ABB RobotStudio station: welding_of_volumetric_parts.rsstn

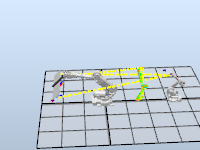
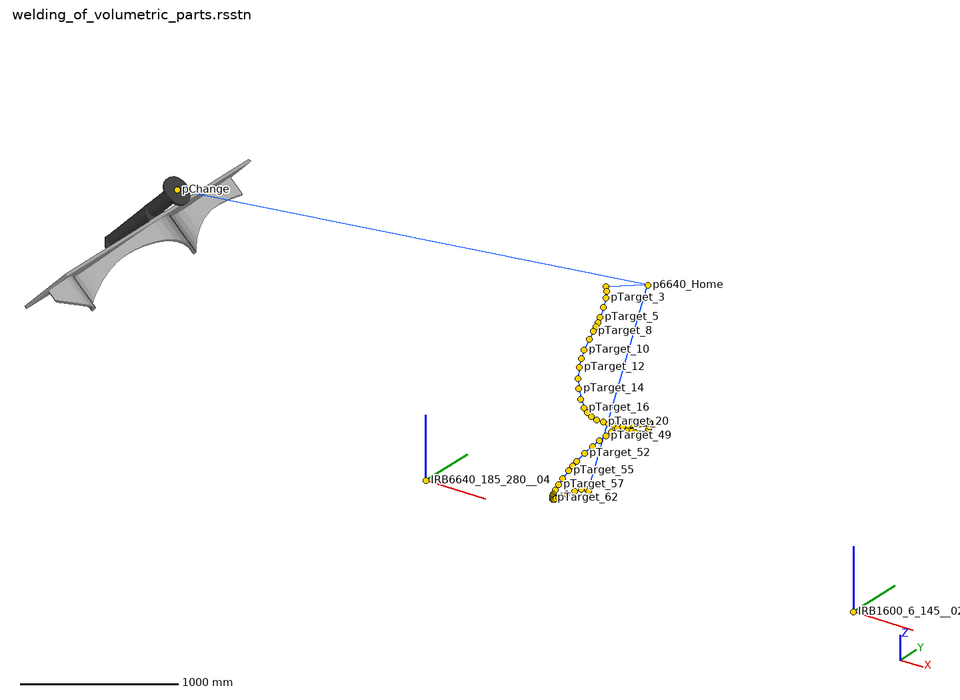
[picture v1: parts stored in the station drawn from their meshes, with robot base, taught points and paths (robot models come from the ABB library and are not in the file)]
Station Station (saved by RobotStudio 21.2.9526.0)
Controller Controller_LR, task T_ROB2: task frame (RAPID world) sits at (3300, 0, 0) mm, rotated rx 0 ry 0 rz 180 deg in the station
Controller Controller_LR, task T_ROB1: task frame (RAPID world) sits at (3300, 0, 0) mm, rotated rx 0 ry 0 rz 180 deg in the station
Controller Controller_LR
  mechanical unit ROB_1: IRB6640_185_280__04, 6 joints, base frame (3300, 0, 0) mm, rotated rx 0 ry 0 rz 180 deg
  mechanical unit ROB_2: IRB1600_6_145__02, 6 joints, base frame (0, 0, 0) mm
Layout (positions relative to the parent item):
  - IRB1600_6_145__02 [mechanism, from Robots\IRB1600_6_145_G_02.rslib] at (3300, 0, 0) mm, rotated rx 0 ry 0 rz 180 deg; joint values [0, -0.6981, 0, 0, 0.4363, 3.1416] (rad or m)
  - IRB6640_185_280__04 [mechanism, from Robots\IRB6640_185_280_G_04.rslib] at (0, 0, 0) mm; joint values [0, -0.6981, -2.2689, 0, -0.9599, 0] (rad or m)
  - training_part1 [part] at (-1918.49, 0, 1506.92) mm, rotated rx 180 ry -45 rz -180 deg, size 449.3 x 2022.8 x 720 mm
  - Binzel_air_22 [mechanism, from Tools\Binzel_air_22.rslib] at (3077.54, 0, 1425.23) mm, rotated rx 0 ry -75 rz 0 deg
Attachment: training_part1 is attached to IRB6640_185_280__04 / Link6
Attachment: Binzel_air_22 is attached to IRB1600_6_145__02 / Link6
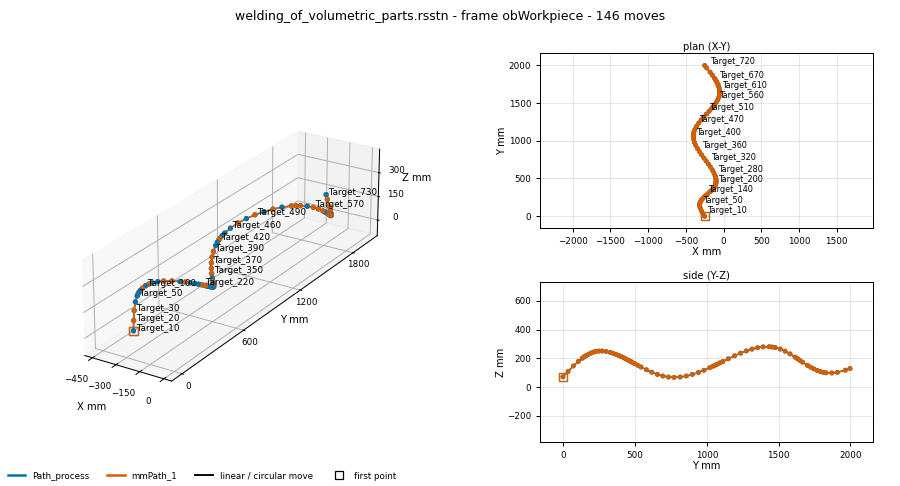
[picture p0: tool path of welding_of_volumetric_parts.rsstn in frame obWorkpiece, 146 of 224 moves have a stored position in this frame; points joined in program order, loops and branches not executed]
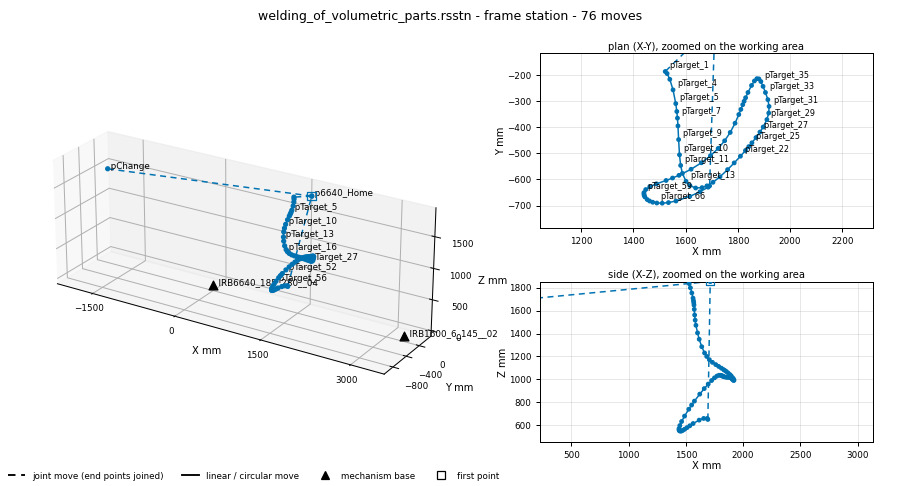
[picture p1: tool path of welding_of_volumetric_parts.rsstn in frame station, 76 of 224 moves have a stored position in this frame; points joined in program order, loops and branches not executed]
Targets, tools, work objects and paths stored in the station, written as RAPID:
! task T_ROB1
MODULE Module1
  VAR SyncIdent Ident_1;
  VAR SyncIdent Ident_2;
  PERS Tasks Task_1{2}:=[["T_ROB1"],["T_ROB2"]];
  CONST robtarget pTarget_1:=[[1778.181697527,186.200299858,1862.655645301],[0.542148406,0.793411995,0.256756469,-0.103192188],[-1,0,-1,0],[9E+09,9E+09,9E+09,9E+09,9E+09,9E+09]];
  CONST robtarget pTarget_2:=[[1770.994188299,194.050467885,1836.295876308],[0.547547156,0.793734178,0.24715111,-0.095365067],[-1,0,-1,0],[9E+09,9E+09,9E+09,9E+09,9E+09,9E+09]];
  CONST robtarget pTarget_3:=[[1760.652825255,216.161560279,1800.133289507],[0.558555641,0.792378,0.228049318,-0.090256356],[-1,0,-1,0],[9E+09,9E+09,9E+09,9E+09,9E+09,9E+09]];
  CONST robtarget pTarget_4:=[[1748.290299895,256.657627996,1755.126396139],[0.576885547,0.787168315,0.198285168,-0.090841082],[-1,0,-1,0],[9E+09,9E+09,9E+09,9E+09,9E+09,9E+09]];
  CONST robtarget pTarget_5:=[[1737.829387141,309.266346265,1710.003660644],[0.600170273,0.776755771,0.163693874,-0.098236606],[-1,0,-1,0],[9E+09,9E+09,9E+09,9E+09,9E+09,9E+09]];
  CONST robtarget pTarget_6:=[[1733.804937068,339.397116728,1687.439781271],[0.613523349,0.769208972,0.145104916,-0.104169199],[-1,0,-1,0],[9E+09,9E+09,9E+09,9E+09,9E+09,9E+09]];
  CONST robtarget pTarget_7:=[[1731.345474568,364.887069734,1669.469926767],[0.624865432,0.761982746,0.12988239,-0.109800051],[-1,0,-1,0],[9E+09,9E+09,9E+09,9E+09,9E+09,9E+09]];
  CONST robtarget pTarget_8:=[[1729.439217622,394.798254229,1649.227463455],[0.638246376,0.752542699,0.112494045,-0.116902268],[-1,0,-1,0],[9E+09,9E+09,9E+09,9E+09,9E+09,9E+09]];
  CONST robtarget pTarget_9:=[[1726.894203356,447.184397046,1611.766562004],[0.661982515,0.733744338,0.082051113,-0.129096907],[-1,0,-1,0],[9E+09,9E+09,9E+09,9E+09,9E+09,9E+09]];
  CONST robtarget pTarget_10:=[[1723.544484943,505.45769037,1562.230464943],[0.689273971,0.709178686,0.04680241,-0.140629006],[-1,0,-1,0],[9E+09,9E+09,9E+09,9E+09,9E+09,9E+09]];
  CONST robtarget pTarget_11:=[[1719.097770684,546.281247526,1517.405345945],[0.709465359,0.689213309,0.019587314,-0.145808972],[-1,0,-1,0],[9E+09,9E+09,9E+09,9E+09,9E+09,9E+09]];
  CONST robtarget pTarget_12:=[[1712.357728352,576.685538105,1472.436688768],[0.725592454,0.672374376,-0.004172996,-0.146324552],[-1,0,-1,0],[9E+09,9E+09,9E+09,9E+09,9E+09,9E+09]];
  CONST robtarget pTarget_13:=[[1698.481718308,607.168067285,1406.157920867],[0.743150521,0.65316553,-0.03513516,-0.140952521],[-1,1,-1,0],[9E+09,9E+09,9E+09,9E+09,9E+09,9E+09]];
  CONST robtarget pTarget_14:=[[1683.689245608,623.318514853,1350.511714032],[0.752710379,0.642114247,-0.059185356,-0.132715759],[-1,1,-1,0],[9E+09,9E+09,9E+09,9E+09,9E+09,9E+09]];
  CONST robtarget pTarget_15:=[[1661.611102892,632.661072606,1285.206196443],[0.756964574,0.636483122,-0.086573404,-0.119995478],[-1,1,-1,0],[9E+09,9E+09,9E+09,9E+09,9E+09,9E+09]];
  CONST robtarget pTarget_16:=[[1636.974570689,631.269638782,1230.880629936],[0.752461483,0.640504386,-0.109446392,-0.107598031],[-1,1,-1,0],[9E+09,9E+09,9E+09,9E+09,9E+09,9E+09]];
  CONST robtarget pTarget_17:=[[1618.266585822,624.412772296,1200.303251277],[0.744570861,0.648569679,-0.122376791,-0.099977627],[-1,1,-1,0],[9E+09,9E+09,9E+09,9E+09,9E+09,9E+09]];
  CONST robtarget pTarget_18:=[[1595.31025739,610.899403989,1172.356577935],[0.73138813,0.662260205,-0.133827929,-0.092590006],[-1,0,-1,0],[9E+09,9E+09,9E+09,9E+09,9E+09,9E+09]];
  CONST robtarget pTarget_19:=[[1568.252391964,589.541208244,1148.621347281],[0.712476477,0.681687181,-0.142360657,-0.086100519],[-1,0,-1,0],[9E+09,9E+09,9E+09,9E+09,9E+09,9E+09]];
  CONST robtarget pTarget_20:=[[1539.248164994,562.206507767,1129.084627739],[0.689417374,0.704583469,-0.14724324,-0.081149543],[-1,0,-1,0],[9E+09,9E+09,9E+09,9E+09,9E+09,9E+09]];
  CONST robtarget pTarget_21:=[[1513.907722067,536.515023967,1113.043516835],[0.667709522,0.725077896,-0.149409413,-0.078120848],[-1,0,-1,0],[9E+09,9E+09,9E+09,9E+09,9E+09,9E+09]];
  CONST robtarget pTarget_22:=[[1490.06843077,510.919096367,1097.932249558],[0.645797019,0.744781689,-0.14976235,-0.076273744],[-1,0,-1,0],[9E+09,9E+09,9E+09,9E+09,9E+09,9E+09]];
  CONST robtarget pTarget_23:=[[1470.694976412,489.03192048,1085.160534616],[0.626718168,0.761182635,-0.148768738,-0.075453277],[-1,0,-1,0],[9E+09,9E+09,9E+09,9E+09,9E+09,9E+09]];
  CONST robtarget pTarget_24:=[[1458.007723014,474.098201767,1076.33725701],[0.613483711,0.772169291,-0.1474183,-0.075234082],[-1,0,-1,0],[9E+09,9E+09,9E+09,9E+09,9E+09,9E+09]];
  CONST robtarget pTarget_25:=[[1446.078098007,459.539371712,1067.555038967],[0.600400247,0.7827328,-0.145556297,-0.075248068],[-1,0,-1,0],[9E+09,9E+09,9E+09,9E+09,9E+09,9E+09]];
  CONST robtarget pTarget_26:=[[1430.366054644,439.373713996,1054.998732884],[0.581991211,0.79712615,-0.142004112,-0.075570919],[-1,0,-1,0],[9E+09,9E+09,9E+09,9E+09,9E+09,9E+09]];
  CONST robtarget pTarget_27:=[[1415.237180171,418.35370749,1041.410054838],[0.562513897,0.811812528,-0.136879951,-0.076173582],[-1,0,-1,0],[9E+09,9E+09,9E+09,9E+09,9E+09,9E+09]];
  CONST robtarget pTarget_28:=[[1402.771915738,398.850948614,1028.566708002],[0.544352217,0.825073539,-0.130500397,-0.076837271],[-1,0,-1,0],[9E+09,9E+09,9E+09,9E+09,9E+09,9E+09]];
  CONST robtarget pTarget_29:=[[1388.675746224,370.620414979,1010.850537495],[0.51852618,0.843366276,-0.117612802,-0.077660507],[-1,0,-1,0],[9E+09,9E+09,9E+09,9E+09,9E+09,9E+09]];
  CONST robtarget pTarget_30:=[[1381.505127476,345.421826654,998.208633001],[0.496784489,0.858370646,-0.101553477,-0.0780506],[-1,0,-1,0],[9E+09,9E+09,9E+09,9E+09,9E+09,9E+09]];
  CONST robtarget pTarget_31:=[[1380.290516089,319.995796425,991.083428878],[0.476896608,0.871763761,-0.08058855,-0.078122058],[-1,0,-1,0],[9E+09,9E+09,9E+09,9E+09,9E+09,9E+09]];
  CONST robtarget pTarget_32:=[[1384.804951043,294.079129956,991.316325422],[0.459310049,0.883135387,-0.054791455,-0.078128501],[-1,0,-1,0],[9E+09,9E+09,9E+09,9E+09,9E+09,9E+09]];
  CONST robtarget pTarget_33:=[[1394.1525823,266.790336369,999.873922559],[0.444147512,0.892188142,-0.024126684,-0.078429645],[-1,0,-1,0],[9E+09,9E+09,9E+09,9E+09,9E+09,9E+09]];
  CONST robtarget pTarget_34:=[[1403.35211698,243.260443714,1008.918127426],[0.434369588,0.897321439,0.002999803,-0.078283439],[-1,0,-1,0],[9E+09,9E+09,9E+09,9E+09,9E+09,9E+09]];
  CONST robtarget pTarget_35:=[[1411.682544208,224.637178453,1015.29477329],[0.430285328,0.899008786,0.024823279,-0.077598603],[-1,0,-1,0],[9E+09,9E+09,9E+09,9E+09,9E+09,9E+09]];
  CONST robtarget pTarget_36:=[[1419.11003976,214.609895019,1018.179510145],[0.432472832,0.89755412,0.037974746,-0.07695303],[-1,0,-1,0],[9E+09,9E+09,9E+09,9E+09,9E+09,9E+09]];
  CONST robtarget pTarget_37:=[[1426.951902197,213.764025906,1018.6233173],[0.440284983,0.893530289,0.042798746,-0.076948195],[-1,0,-1,0],[9E+09,9E+09,9E+09,9E+09,9E+09,9E+09]];
  CONST robtarget pTarget_38:=[[1436.38652418,222.488667703,1018.14305052],[0.453338467,0.88700135,0.039811537,-0.078280782],[-1,0,-1,0],[9E+09,9E+09,9E+09,9E+09,9E+09,9E+09]];
  CONST robtarget pTarget_39:=[[1447.431300545,239.694255611,1018.408583383],[0.470271988,0.878223745,0.030346137,-0.081525599],[-1,0,-1,0],[9E+09,9E+09,9E+09,9E+09,9E+09,9E+09]];
  CONST robtarget pTarget_40:=[[1461.186292661,266.637925532,1021.027640653],[0.492377698,0.865821477,0.014387778,-0.087808685],[-1,0,-1,0],[9E+09,9E+09,9E+09,9E+09,9E+09,9E+09]];
  CONST robtarget pTarget_41:=[[1470.20295235,286.708972067,1024.274155825],[0.507484444,0.85659197,0.002382892,-0.093295538],[-1,0,-1,0],[9E+09,9E+09,9E+09,9E+09,9E+09,9E+09]];
  CONST robtarget pTarget_42:=[[1475.847241271,300.225934757,1026.972648038],[0.517297415,0.850233009,-0.005676712,-0.097339556],[-1,0,-1,0],[9E+09,9E+09,9E+09,9E+09,9E+09,9E+09]];
  CONST robtarget pTarget_43:=[[1481.114497039,313.307838348,1029.67109328],[0.526490151,0.84400693,-0.013395766,-0.101395152],[-1,0,-1,0],[9E+09,9E+09,9E+09,9E+09,9E+09,9E+09]];
  CONST robtarget pTarget_44:=[[1488.33776285,331.436834376,1032.939801302],[0.538604529,0.835396873,-0.023911904,-0.106983393],[-1,0,-1,0],[9E+09,9E+09,9E+09,9E+09,9E+09,9E+09]];
  CONST robtarget pTarget_45:=[[1496.282697007,351.178665453,1035.489566541],[0.550971738,0.826113149,-0.035175987,-0.112826679],[-1,0,-1,0],[9E+09,9E+09,9E+09,9E+09,9E+09,9E+09]];
  CONST robtarget pTarget_46:=[[1510.659226816,384.392866719,1035.936669737],[0.569767124,0.811017832,-0.053856936,-0.121305115],[-1,0,-1,0],[9E+09,9E+09,9E+09,9E+09,9E+09,9E+09]];
  CONST robtarget pTarget_47:=[[1529.151843225,419.773837395,1028.594126136],[0.586873423,0.796247642,-0.073737743,-0.127011905],[-1,0,-1,0],[9E+09,9E+09,9E+09,9E+09,9E+09,9E+09]];
  CONST robtarget pTarget_48:=[[1550.527278537,451.696712634,1013.011343794],[0.599817679,0.784445953,-0.092153229,-0.127949526],[-1,0,-1,0],[9E+09,9E+09,9E+09,9E+09,9E+09,9E+09]];
  CONST robtarget pTarget_49:=[[1575.38815922,481.045847154,990.004702603],[0.609952056,0.774798228,-0.110108005,-0.124589014],[-1,0,-1,0],[9E+09,9E+09,9E+09,9E+09,9E+09,9E+09]];
  CONST robtarget pTarget_50:=[[1605.096587084,509.301137558,958.828336985],[0.618413471,0.766286888,-0.129146859,-0.117005441],[-1,0,-1,0],[9E+09,9E+09,9E+09,9E+09,9E+09,9E+09]];
  CONST robtarget pTarget_51:=[[1639.809434498,536.118324815,919.166331526],[0.625325492,0.75856786,-0.149973283,-0.105123002],[-1,0,-1,0],[9E+09,9E+09,9E+09,9E+09,9E+09,9E+09]];
  CONST robtarget pTarget_52:=[[1679.199810422,560.815010805,870.890635487],[0.630309247,0.751520378,-0.173247334,-0.08895356],[-1,0,-1,0],[9E+09,9E+09,9E+09,9E+09,9E+09,9E+09]];
  CONST robtarget pTarget_53:=[[1725.528962599,584.086235135,809.910787471],[0.632355869,0.744936605,-0.201701212,-0.067172388],[-1,0,-1,0],[9E+09,9E+09,9E+09,9E+09,9E+09,9E+09]];
  CONST robtarget pTarget_54:=[[1750.172428429,594.482484706,775.388290642],[0.63140608,0.7421901,-0.217958794,-0.054536053],[-1,0,-1,0],[9E+09,9E+09,9E+09,9E+09,9E+09,9E+09]];
  CONST robtarget pTarget_55:=[[1774.856620893,603.840371659,738.910588443],[0.628566044,0.740077047,-0.235575569,-0.041168483],[-1,0,-1,0],[9E+09,9E+09,9E+09,9E+09,9E+09,9E+09]];
  CONST robtarget pTarget_56:=[[1811.777191977,616.730180478,679.050006644],[0.618911201,0.738755968,-0.266073975,-0.019828897],[-1,0,-1,0],[9E+09,9E+09,9E+09,9E+09,9E+09,9E+09]];
  CONST robtarget pTarget_57:=[[1837.481090124,627.77802117,631.687814205],[0.602922247,0.74259699,-0.291560622,-0.005184429],[-1,0,-1,0],[9E+09,9E+09,9E+09,9E+09,9E+09,9E+09]];
  CONST robtarget pTarget_58:=[[1853.13231236,638.757228397,596.097182329],[0.580906923,0.752194854,-0.311036519,0.002516262],[-1,0,-1,0],[9E+09,9E+09,9E+09,9E+09,9E+09,9E+09]];
  CONST robtarget pTarget_59:=[[1859.687990898,650.495043313,570.285600703],[0.552220417,0.768070307,-0.324202492,0.003654924],[-1,0,-1,0],[9E+09,9E+09,9E+09,9E+09,9E+09,9E+09]];
  CONST robtarget pTarget_60:=[[1859.811053846,656.41145748,561.173098787],[0.536445912,0.777595711,-0.32797363,0.001997943],[-1,0,-1,0],[9E+09,9E+09,9E+09,9E+09,9E+09,9E+09]];
  CONST robtarget pTarget_61:=[[1858.736717823,661.312610851,555.257299322],[0.52319042,0.785855215,-0.329701861,-0.000220179],[-1,0,-1,0],[9E+09,9E+09,9E+09,9E+09,9E+09,9E+09]];
  CONST robtarget pTarget_62:=[[1856.112823082,667.023889107,550.266827904],[0.507419782,0.796023651,-0.329935382,-0.003762518],[-1,0,-1,0],[9E+09,9E+09,9E+09,9E+09,9E+09,9E+09]];
  CONST robtarget pTarget_63:=[[1847.230721406,676.928437841,547.055177598],[0.478317899,0.815833575,-0.324757713,-0.012648867],[-1,0,-1,0],[9E+09,9E+09,9E+09,9E+09,9E+09,9E+09]];
  CONST robtarget pTarget_64:=[[1838.321156584,682.542587842,549.276490839],[0.459490769,0.829323493,-0.317325526,-0.019881854],[-1,0,-1,0],[9E+09,9E+09,9E+09,9E+09,9E+09,9E+09]];
  CONST robtarget pTarget_65:=[[1826.161173726,687.193934661,555.142376291],[0.440225806,0.843543883,-0.306320812,-0.028328734],[-1,0,-1,0],[9E+09,9E+09,9E+09,9E+09,9E+09,9E+09]];
  CONST robtarget pTarget_66:=[[1810.310361427,690.231237949,564.749774935],[0.420856439,0.85808964,-0.291782518,-0.037749037],[-1,0,-1,0],[9E+09,9E+09,9E+09,9E+09,9E+09,9E+09]];
  CONST robtarget pTarget_67:=[[1789.773552916,690.927456877,578.389598935],[0.401138523,0.872938401,-0.273398943,-0.04816068],[-1,0,-1,0],[9E+09,9E+09,9E+09,9E+09,9E+09,9E+09]];
  CONST robtarget pTarget_68:=[[1765.75021051,688.568865454,594.763074341],[0.382661443,0.886685714,-0.252838714,-0.058576872],[-1,0,-1,0],[9E+09,9E+09,9E+09,9E+09,9E+09,9E+09]];
  CONST robtarget pTarget_69:=[[1737.046563543,682.522254093,614.005661637],[0.364576903,0.899759243,-0.229606282,-0.069267178],[-1,0,-1,0],[9E+09,9E+09,9E+09,9E+09,9E+09,9E+09]];
  CONST robtarget pTarget_70:=[[1684.060962191,664.78186504,643.84125629],[0.336296246,0.918529025,-0.18976067,-0.084853721],[-1,0,-1,0],[9E+09,9E+09,9E+09,9E+09,9E+09,9E+09]];
  CONST robtarget pTarget_71:=[[1645.011621204,647.158478783,658.508174855],[0.317990031,0.929509253,-0.162018372,-0.092978151],[-1,0,-1,0],[9E+09,9E+09,9E+09,9E+09,9E+09,9E+09]];
  CONST robtarget pTarget_72:=[[1613.795609877,629.560102821,658.605457436],[0.303529417,0.937801267,-0.138776902,-0.095601507],[-1,0,-1,0],[9E+09,9E+09,9E+09,9E+09,9E+09,9E+09]];
  CONST robtarget pTarget_73:=[[1608.138872873,624.65265311,649.727513322],[0.299609152,0.940249896,-0.132011271,-0.093474667],[-1,0,-1,0],[9E+09,9E+09,9E+09,9E+09,9E+09,9E+09]];
  CONST robtarget p6640_Home:=[[1587.499974331,-0.000006468,1854.999955426],[-0.000000016,1,0.000000016,0.000000038],[0,0,-1,0],[9E+09,9E+09,9E+09,9E+09,9E+09,9E+09]];
  CONST robtarget pChange:=[[5218.492492903,0.000005298,1506.919831082],[0.00000001,0.923879547,0.000000011,0.382683398],[-1,0,-1,7],[9E+09,9E+09,9E+09,9E+09,9E+09,9E+09]];
  PROC mmPath_1()
    MoveJ p6640_Home,v1000,z100,tool0\WObj:=wobj0;
    SyncMoveOn Ident_1,Task_1;
    MoveJ pTarget_1\ID:=10,v1000,z100,tool0\WObj:=wobj0;
    MoveL pTarget_2\ID:=20,v1000,z100,tool0\WObj:=wobj0;
    MoveL pTarget_3\ID:=30,v1000,z100,tool0\WObj:=wobj0;
    MoveL pTarget_4\ID:=40,v1000,z100,tool0\WObj:=wobj0;
    MoveL pTarget_5\ID:=50,v1000,z100,tool0\WObj:=wobj0;
    MoveL pTarget_6\ID:=60,v1000,z100,tool0\WObj:=wobj0;
    MoveL pTarget_7\ID:=70,v1000,z100,tool0\WObj:=wobj0;
    MoveL pTarget_8\ID:=80,v1000,z100,tool0\WObj:=wobj0;
    MoveL pTarget_9\ID:=90,v1000,z100,tool0\WObj:=wobj0;
    MoveL pTarget_10\ID:=100,v1000,z100,tool0\WObj:=wobj0;
    MoveL pTarget_11\ID:=110,v1000,z100,tool0\WObj:=wobj0;
    MoveL pTarget_12\ID:=120,v1000,z100,tool0\WObj:=wobj0;
    MoveL pTarget_13\ID:=130,v1000,z100,tool0\WObj:=wobj0;
    MoveL pTarget_14\ID:=140,v1000,z100,tool0\WObj:=wobj0;
    MoveL pTarget_15\ID:=150,v1000,z100,tool0\WObj:=wobj0;
    MoveL pTarget_16\ID:=160,v1000,z100,tool0\WObj:=wobj0;
    MoveL pTarget_17\ID:=170,v1000,z100,tool0\WObj:=wobj0;
    MoveL pTarget_18\ID:=180,v1000,z100,tool0\WObj:=wobj0;
    MoveL pTarget_19\ID:=190,v1000,z100,tool0\WObj:=wobj0;
    MoveL pTarget_20\ID:=200,v1000,z100,tool0\WObj:=wobj0;
    MoveL pTarget_21\ID:=210,v1000,z100,tool0\WObj:=wobj0;
    MoveL pTarget_22\ID:=220,v1000,z100,tool0\WObj:=wobj0;
    MoveL pTarget_23\ID:=230,v1000,z100,tool0\WObj:=wobj0;
    MoveL pTarget_24\ID:=240,v1000,z100,tool0\WObj:=wobj0;
    MoveL pTarget_25\ID:=250,v1000,z100,tool0\WObj:=wobj0;
    MoveL pTarget_26\ID:=260,v1000,z100,tool0\WObj:=wobj0;
    MoveL pTarget_27\ID:=270,v1000,z100,tool0\WObj:=wobj0;
    MoveL pTarget_28\ID:=280,v1000,z100,tool0\WObj:=wobj0;
    MoveL pTarget_29\ID:=290,v1000,z100,tool0\WObj:=wobj0;
    MoveL pTarget_30\ID:=300,v1000,z100,tool0\WObj:=wobj0;
    MoveL pTarget_31\ID:=310,v1000,z100,tool0\WObj:=wobj0;
    MoveL pTarget_32\ID:=320,v1000,z100,tool0\WObj:=wobj0;
    MoveL pTarget_33\ID:=330,v1000,z100,tool0\WObj:=wobj0;
    MoveL pTarget_34\ID:=340,v1000,z100,tool0\WObj:=wobj0;
    MoveL pTarget_35\ID:=350,v1000,z100,tool0\WObj:=wobj0;
    MoveL pTarget_36\ID:=360,v1000,z100,tool0\WObj:=wobj0;
    MoveL pTarget_37\ID:=370,v1000,z100,tool0\WObj:=wobj0;
    MoveL pTarget_38\ID:=380,v1000,z100,tool0\WObj:=wobj0;
    MoveL pTarget_39\ID:=390,v1000,z100,tool0\WObj:=wobj0;
    MoveL pTarget_40\ID:=400,v1000,z100,tool0\WObj:=wobj0;
    MoveL pTarget_41\ID:=410,v1000,z100,tool0\WObj:=wobj0;
    MoveL pTarget_42\ID:=420,v1000,z100,tool0\WObj:=wobj0;
    MoveL pTarget_43\ID:=430,v1000,z100,tool0\WObj:=wobj0;
    MoveL pTarget_44\ID:=440,v1000,z100,tool0\WObj:=wobj0;
    MoveL pTarget_45\ID:=450,v1000,z100,tool0\WObj:=wobj0;
    MoveL pTarget_46\ID:=460,v1000,z100,tool0\WObj:=wobj0;
    MoveL pTarget_47\ID:=470,v1000,z100,tool0\WObj:=wobj0;
    MoveL pTarget_48\ID:=480,v1000,z100,tool0\WObj:=wobj0;
    MoveL pTarget_49\ID:=490,v1000,z100,tool0\WObj:=wobj0;
    MoveL pTarget_50\ID:=500,v1000,z100,tool0\WObj:=wobj0;
    MoveL pTarget_51\ID:=510,v1000,z100,tool0\WObj:=wobj0;
    MoveL pTarget_52\ID:=520,v1000,z100,tool0\WObj:=wobj0;
    MoveL pTarget_53\ID:=530,v1000,z100,tool0\WObj:=wobj0;
    MoveL pTarget_54\ID:=540,v1000,z100,tool0\WObj:=wobj0;
    MoveL pTarget_55\ID:=550,v1000,z100,tool0\WObj:=wobj0;
    MoveL pTarget_56\ID:=560,v1000,z100,tool0\WObj:=wobj0;
    MoveL pTarget_57\ID:=570,v1000,z100,tool0\WObj:=wobj0;
    MoveL pTarget_58\ID:=580,v1000,z100,tool0\WObj:=wobj0;
    MoveL pTarget_59\ID:=590,v1000,z100,tool0\WObj:=wobj0;
    MoveL pTarget_60\ID:=600,v1000,z100,tool0\WObj:=wobj0;
    MoveL pTarget_61\ID:=610,v1000,z100,tool0\WObj:=wobj0;
    MoveL pTarget_62\ID:=620,v1000,z100,tool0\WObj:=wobj0;
    MoveL pTarget_63\ID:=630,v1000,z100,tool0\WObj:=wobj0;
    MoveL pTarget_64\ID:=640,v1000,z100,tool0\WObj:=wobj0;
    MoveL pTarget_65\ID:=650,v1000,z100,tool0\WObj:=wobj0;
    MoveL pTarget_66\ID:=660,v1000,z100,tool0\WObj:=wobj0;
    MoveL pTarget_67\ID:=670,v1000,z100,tool0\WObj:=wobj0;
    MoveL pTarget_68\ID:=680,v1000,z100,tool0\WObj:=wobj0;
    MoveL pTarget_69\ID:=690,v1000,z100,tool0\WObj:=wobj0;
    MoveL pTarget_70\ID:=700,v1000,z100,tool0\WObj:=wobj0;
    MoveL pTarget_71\ID:=710,v1000,z100,tool0\WObj:=wobj0;
    MoveL pTarget_72\ID:=720,v1000,z100,tool0\WObj:=wobj0;
    MoveL pTarget_73\ID:=730,v1000,fine,tool0\WObj:=wobj0;
    SyncMoveOff Ident_2;
    MoveJ p6640_Home,v1000,z100,tool0\WObj:=wobj0;
    MoveJ pChange,v1000,z100,tool0\WObj:=wobj0;
  ENDPROC
  PROC main()
    mmPath_1;
  ENDPROC
ENDMODULE

! task T_ROB2
MODULE CalibData
  PERS tooldata tWeldGun:=[TRUE,[[125.800591275,0,391.268161315],[0.898794046,0,0.438371147,0]],[3,[0,0,100],[0,1,0,0],0,0,0]];
  TASK PERS wobjdata obWorkpiece:=[FALSE,FALSE,"ROB_1",[[755.757189853,1010,1655.621671169],[-0.00000031,-0.258821852,0.000001158,0.965925074]],[[-69.999626585,-1010,719.999567418],[0.707108836,0.000000311,-0.707104726,0.000001158]]];
ENDMODULE

! task T_ROB2
MODULE Module1
  CONST robtarget Target_10:=[[-249.999982853,-2.758889972,70.910184906],[0.218727356,-0.500318169,-0.767608398,-0.335585192],[0,0,0,0],[9E+09,9E+09,9E+09,9E+09,9E+09,9E+09]];
  CONST robtarget Target_20:=[[-272.861882141,33.004474389,109.271780859],[0.218070089,-0.506815721,-0.766106922,-0.329641389],[0,0,0,0],[9E+09,9E+09,9E+09,9E+09,9E+09,9E+09]];
  CONST robtarget Target_30:=[[-293.910897367,69.704818109,146.788417202],[0.216170638,-0.529374655,-0.759500655,-0.31014752],[0,0,0,0],[9E+09,9E+09,9E+09,9E+09,9E+09,9E+09]];
  CONST robtarget Target_40:=[[-309.050426556,104.288383302,178.815114444],[0.21342224,-0.572774596,-0.741629436,-0.276343968],[0,0,0,0],[9E+09,9E+09,9E+09,9E+09,9E+09,9E+09]];
  CONST robtarget Target_50:=[[-315.825879092,131.080277492,200.511993969],[0.210053721,-0.629622145,-0.709520967,-0.236713724],[0,0,0,0],[9E+09,9E+09,9E+09,9E+09,9E+09,9E+09]];
  CONST robtarget Target_60:=[[-316.950658169,142.443127526,208.736277874],[0.207697142,-0.661844648,-0.687247207,-0.215672981],[0,0,0,0],[9E+09,9E+09,9E+09,9E+09,9E+09,9E+09]];
  CONST robtarget Target_70:=[[-316.982935585,150.772590841,214.3610347],[0.205252938,-0.688776438,-0.666352974,-0.198574832],[0,0,0,0],[9E+09,9E+09,9E+09,9E+09,9E+09,9E+09]];
  CONST robtarget Target_80:=[[-316.205680892,159.554683635,219.903696352],[0.201637265,-0.719895206,-0.63953479,-0.179132795],[0,0,0,0],[9E+09,9E+09,9E+09,9E+09,9E+09,9E+09]];
  CONST robtarget Target_90:=[[-312.752948072,174.804783132,228.537464358],[0.190111882,-0.772966578,-0.58777574,-0.144567705],[0,0,0,0],[9E+09,9E+09,9E+09,9E+09,9E+09,9E+09]];
  CONST robtarget Target_100:=[[-304.930214203,193.592151989,237.349035256],[0.164735755,-0.829787877,-0.523003524,-0.10383412],[0,0,0,0],[9E+09,9E+09,9E+09,9E+09,9E+09,9E+09]];
  CONST robtarget Target_110:=[[-295.354295578,209.583594983,243.175290065],[0.133385277,-0.8681553,-0.472487419,-0.0725974],[0,0,0,0],[9E+09,9E+09,9E+09,9E+09,9E+09,9E+09]];
  CONST robtarget Target_120:=[[-283.899433589,224.892894657,247.248273661],[0.09596897,-0.895792145,-0.43151926,-0.046233299],[0,0,0,0],[9E+09,9E+09,9E+09,9E+09,9E+09,9E+09]];
  CONST robtarget Target_130:=[[-263.241026813,247.749218638,250.55023108],[0.034733915,-0.921371183,-0.386853892,-0.014586439],[0,0,0,0],[9E+09,9E+09,9E+09,9E+09,9E+09,9E+09]];
  CONST robtarget Target_140:=[[-240.981922532,269.119698062,250.907521043],[0.018476819,0.931695715,0.362698235,-0.007189718],[0,0,0,0],[9E+09,9E+09,9E+09,9E+09,9E+09,9E+09]];
  CONST robtarget Target_150:=[[-208.413183072,298.032091366,247.788399876],[0.079579938,0.931527315,0.353569956,-0.030202349],[0,0,0,0],[9E+09,9E+09,9E+09,9E+09,9E+09,9E+09]];
  CONST robtarget Target_160:=[[-176.052193628,326.809908438,241.224111838],[0.12634207,0.919491885,0.3687884,-0.050670216],[0,0,0,0],[9E+09,9E+09,9E+09,9E+09,9E+09,9E+09]];
  CONST robtarget Target_170:=[[-156.253006236,345.812062065,235.319898524],[0.149532826,0.905306343,0.392253601,-0.0647879],[0,0,0,0],[9E+09,9E+09,9E+09,9E+09,9E+09,9E+09]];
  CONST robtarget Target_180:=[[-137.912729763,365.729836666,228.01394112],[0.167326436,0.883813043,0.429269038,-0.081267835],[0,0,0,0],[9E+09,9E+09,9E+09,9E+09,9E+09,9E+09]];
  CONST robtarget Target_190:=[[-123.076086452,385.29684741,219.899751042],[0.178122742,0.85378951,0.478888901,-0.099905866],[0,0,0,0],[9E+09,9E+09,9E+09,9E+09,9E+09,9E+09]];
  CONST robtarget Target_200:=[[-112.485109992,403.753339887,211.517517208],[0.182306761,0.816637689,0.534446355,-0.119307265],[0,0,0,0],[9E+09,9E+09,9E+09,9E+09,9E+09,9E+09]];
  CONST robtarget Target_210:=[[-105.670178268,420.540737418,203.413907188],[0.182491022,0.780616625,0.582081066,-0.136074774],[0,0,0,0],[9E+09,9E+09,9E+09,9E+09,9E+09,9E+09]];
  CONST robtarget Target_220:=[[-101.15368719,437.795748992,194.701831653],[0.179971611,0.74337611,0.626119394,-0.151580612],[0,0,0,0],[9E+09,9E+09,9E+09,9E+09,9E+09,9E+09]];
  CONST robtarget Target_230:=[[-99.004909593,453.550262222,186.488207379],[0.175916518,0.71039217,0.661486962,-0.163802752],[0,0,0,0],[9E+09,9E+09,9E+09,9E+09,9E+09,9E+09]];
  CONST robtarget Target_240:=[[-98.517183319,465.110586386,180.346452198],[0.172174243,0.687303096,0.684519732,-0.171473672],[0,0,0,0],[9E+09,9E+09,9E+09,9E+09,9E+09,9E+09]];
  CONST robtarget Target_250:=[[-98.914532644,477.216281927,173.843762862],[0.167750144,0.664394684,0.706153116,-0.178290128],[0,0,0,0],[9E+09,9E+09,9E+09,9E+09,9E+09,9E+09]];
  CONST robtarget Target_260:=[[-101.159356556,495.695093883,163.844728445],[0.160294978,0.632212446,0.734783022,-0.186297754],[0,0,0,0],[9E+09,9E+09,9E+09,9E+09,9E+09,9E+09]];
  CONST robtarget Target_270:=[[-106.105437701,517.567072003,152.023011482],[0.150752486,0.598596041,0.762916676,-0.192131759],[0,0,0,0],[9E+09,9E+09,9E+09,9E+09,9E+09,9E+09]];
  CONST robtarget Target_280:=[[-113.660661173,540.614926982,139.756423783],[0.140145495,0.568163603,0.787297941,-0.194194007],[0,0,0,0],[9E+09,9E+09,9E+09,9E+09,9E+09,9E+09]];
  CONST robtarget Target_290:=[[-130.507634781,578.661910337,120.438432349],[0.121655696,0.527679401,0.819198584,-0.188859792],[0,0,0,0],[9E+09,9E+09,9E+09,9E+09,9E+09,9E+09]];
  CONST robtarget Target_300:=[[-151.26626902,615.99978174,103.274739393],[0.102156402,0.497611338,0.84376747,-0.173215132],[0,0,0,0],[9E+09,9E+09,9E+09,9E+09,9E+09,9E+09]];
  CONST robtarget Target_310:=[[-176.025786598,654.711283406,88.195694778],[0.080012228,0.474620075,0.864351323,-0.1457073],[0,0,0,0],[9E+09,9E+09,9E+09,9E+09,9E+09,9E+09]];
  CONST robtarget Target_320:=[[-202.970062049,693.301100095,76.713070128],[0.055270211,0.458961325,0.880375462,-0.106012978],[0,0,0,0],[9E+09,9E+09,9E+09,9E+09,9E+09,9E+09]];
  CONST robtarget Target_330:=[[-231.601523866,732.417884044,69.538476495],[0.026891104,0.450400962,0.890835712,-0.053174969],[0,0,0,0],[9E+09,9E+09,9E+09,9E+09,9E+09,9E+09]];
  CONST robtarget Target_340:=[[-260.469520449,771.255872105,67.252197805],[0.000040228,0.449762351,0.893148263,-0.000073424],[0,0,0,0],[9E+09,9E+09,9E+09,9E+09,9E+09,9E+09]];
  CONST robtarget Target_350:=[[-291.670914504,813.968978886,69.776506912],[0.026409008,-0.457823003,-0.887175769,-0.051184145],[0,0,0,0],[9E+09,9E+09,9E+09,9E+09,9E+09,9E+09]];
  CONST robtarget Target_360:=[[-321.099734743,856.496080673,76.870467066],[0.050519426,-0.474571222,-0.873828081,-0.093029174],[0,0,0,0],[9E+09,9E+09,9E+09,9E+09,9E+09,9E+09]];
  CONST robtarget Target_370:=[[-347.607513558,898.756689263,87.793598215],[0.073136056,-0.499938347,-0.853878066,-0.124920036],[0,0,0,0],[9E+09,9E+09,9E+09,9E+09,9E+09,9E+09]];
  CONST robtarget Target_380:=[[-370.045783343,940.670316452,101.805420301],[0.094966939,-0.534398849,-0.826923789,-0.146956446],[0,0,0,0],[9E+09,9E+09,9E+09,9E+09,9E+09,9E+09]];
  CONST robtarget Target_390:=[[-386.422266732,979.738715708,117.17043925],[0.115288749,-0.575885363,-0.793612764,-0.15888151],[0,0,0,0],[9E+09,9E+09,9E+09,9E+09,9E+09,9E+09]];
  CONST robtarget Target_400:=[[-397.441208907,1019.683400433,134.627667281],[0.13626385,-0.628500265,-0.748392037,-0.162261943],[0,0,0,0],[9E+09,9E+09,9E+09,9E+09,9E+09,9E+09]];
  CONST robtarget Target_410:=[[-400.684804054,1043.11370182,145.484353571],[0.148540441,-0.664075872,-0.715089643,-0.159955541],[0,0,0,0],[9E+09,9E+09,9E+09,9E+09,9E+09,9E+09]];
  CONST robtarget Target_420:=[[-401.329047191,1057.287009915,152.213033994],[0.155841519,-0.687048546,-0.692119904,-0.156996034],[0,0,0,0],[9E+09,9E+09,9E+09,9E+09,9E+09,9E+09]];
  CONST robtarget Target_430:=[[-400.962324214,1070.626836833,158.630266332],[0.162306824,-0.708452998,-0.669495106,-0.153385619],[0,0,0,0],[9E+09,9E+09,9E+09,9E+09,9E+09,9E+09]];
  CONST robtarget Target_440:=[[-398.849183148,1089.50771848,167.811803441],[0.170245025,-0.736429133,-0.637918276,-0.147475544],[0,0,0,0],[9E+09,9E+09,9E+09,9E+09,9E+09,9E+09]];
  CONST robtarget Target_450:=[[-394.2955253,1110.833995661,178.254456324],[0.177319257,-0.764612398,-0.603598072,-0.139982605],[0,0,0,0],[9E+09,9E+09,9E+09,9E+09,9E+09,9E+09]];
  CONST robtarget Target_460:=[[-380.757471944,1149.009379517,196.873180768],[0.184540979,-0.806336545,-0.547767283,-0.125367489],[0,0,0,0],[9E+09,9E+09,9E+09,9E+09,9E+09,9E+09]];
  CONST robtarget Target_470:=[[-357.502459174,1192.924465348,217.59618262],[0.183790476,-0.842562217,-0.494638737,-0.107900377],[0,0,0,0],[9E+09,9E+09,9E+09,9E+09,9E+09,9E+09]];
  CONST robtarget Target_480:=[[-328.871131996,1234.787325405,235.977961384],[0.173717681,-0.868301552,-0.455593953,-0.091152247],[0,0,0,0],[9E+09,9E+09,9E+09,9E+09,9E+09,9E+09]];
  CONST robtarget Target_490:=[[-297.082271262,1274.589016917,251.512758604],[0.155168267,-0.886933809,-0.428543903,-0.074975664],[0,0,0,0],[9E+09,9E+09,9E+09,9E+09,9E+09,9E+09]];
  CONST robtarget Target_500:=[[-262.487284271,1314.072540843,264.392414029],[0.127341788,-0.900832553,-0.410985687,-0.05809945],[0,0,0,0],[9E+09,9E+09,9E+09,9E+09,9E+09,9E+09]];
  CONST robtarget Target_510:=[[-226.57533141,1353.20491494,273.985918464],[0.089566851,-0.910054777,-0.40274885,-0.039641474],[0,0,0,0],[9E+09,9E+09,9E+09,9E+09,9E+09,9E+09]];
  CONST robtarget Target_520:=[[-190.835573063,1391.953156962,279.66226271],[0.041472362,-0.913491552,-0.404321853,-0.018359371],[0,0,0,0],[9E+09,9E+09,9E+09,9E+09,9E+09,9E+09]];
  CONST robtarget Target_530:=[[-154.17838296,1433.251807008,280.664288166],[0.021076524,0.908000293,0.418326405,-0.009709151],[0,0,0,0],[9E+09,9E+09,9E+09,9E+09,9E+09,9E+09]];
  CONST robtarget Target_540:=[[-136.486765374,1454.464402311,278.839431135],[0.056847305,0.900059217,0.431184714,-0.027231083],[0,0,0,0],[9E+09,9E+09,9E+09,9E+09,9E+09,9E+09]];
  CONST robtarget Target_550:=[[-119.667936085,1475.943296051,275.178359687],[0.094528682,0.887510172,0.448451627,-0.047761511],[0,0,0,0],[9E+09,9E+09,9E+09,9E+09,9E+09,9E+09]];
  CONST robtarget Target_560:=[[-95.234012575,1510.930409762,264.895769368],[0.154652239,0.855971808,0.485490887,-0.087712866],[0,0,0,0],[9E+09,9E+09,9E+09,9E+09,9E+09,9E+09]];
  CONST robtarget Target_570:=[[-75.878773781,1544.776154817,249.922804533],[0.194530976,0.816269054,0.529114868,-0.126095149],[0,0,0,0],[9E+09,9E+09,9E+09,9E+09,9E+09,9E+09]];
  CONST robtarget Target_580:=[[-61.453141161,1578.970333156,230.887297549],[0.213995385,0.770545603,0.578493801,-0.160656062],[0,0,0,0],[9E+09,9E+09,9E+09,9E+09,9E+09,9E+09]];
  CONST robtarget Target_590:=[[-52.708491627,1614.593802629,208.278633282],[0.2154784,0.717600683,0.634304305,-0.190463561],[0,0,0,0],[9E+09,9E+09,9E+09,9E+09,9E+09,9E+09]];
  CONST robtarget Target_600:=[[-50.933702908,1632.587902032,196.272906508],[0.21049827,0.690275184,0.662147881,-0.201917887],[0,0,0,0],[9E+09,9E+09,9E+09,9E+09,9E+09,9E+09]];
  CONST robtarget Target_610:=[[-50.773310022,1647.959263114,185.915184413],[0.204128011,0.668216161,0.684203386,-0.209008715],[0,0,0,0],[9E+09,9E+09,9E+09,9E+09,9E+09,9E+09]];
  CONST robtarget Target_620:=[[-52.133848077,1666.482662645,173.501879979],[0.194191907,0.643165566,0.709079002,-0.214089997],[0,0,0,0],[9E+09,9E+09,9E+09,9E+09,9E+09,9E+09]];
  CONST robtarget Target_630:=[[-58.782669223,1700.877359567,151.375731817],[0.170010517,0.600573609,0.751746936,-0.2128011],[0,0,0,0],[9E+09,9E+09,9E+09,9E+09,9E+09,9E+09]];
  CONST robtarget Target_640:=[[-65.573382217,1722.873059911,138.379981308],[0.151037739,0.575542272,0.777381463,-0.204001853],[0,0,0,0],[9E+09,9E+09,9E+09,9E+09,9E+09,9E+09]];
  CONST robtarget Target_650:=[[-74.172458436,1744.953551809,126.646734635],[0.129487963,0.551841007,0.802051755,-0.188194988],[0,0,0,0],[9E+09,9E+09,9E+09,9E+09,9E+09,9E+09]];
  CONST robtarget Target_660:=[[-84.216406288,1766.689925652,116.694082829],[0.10605041,0.529831854,0.825081517,-0.165142384],[0,0,0,0],[9E+09,9E+09,9E+09,9E+09,9E+09,9E+09]];
  CONST robtarget Target_670:=[[-95.703735197,1788.481494933,108.58929655],[0.080632832,0.509232536,0.84630056,-0.133999749],[0,0,0,0],[9E+09,9E+09,9E+09,9E+09,9E+09,9E+09]];
  CONST robtarget Target_680:=[[-107.611560112,1808.886865418,102.932793062],[0.055430058,0.491624274,0.863570533,-0.097360244],[0,0,0,0],[9E+09,9E+09,9E+09,9E+09,9E+09,9E+09]];
  CONST robtarget Target_690:=[[-120.619803812,1829.451884245,99.303968751],[0.029389138,0.476040843,0.877262115,-0.054153266],[0,0,0,0],[9E+09,9E+09,9E+09,9E+09,9E+09,9E+09]];
  CONST robtarget Target_700:=[[-148.697947715,1869.907233475,98.051310221],[0.01238213,-0.453317439,-0.890930671,-0.024341782],[0,0,0,0],[9E+09,9E+09,9E+09,9E+09,9E+09,9E+09]];
  CONST robtarget Target_710:=[[-178.285867762,1909.003244069,102.928222428],[0.041270541,-0.440304957,-0.892984494,-0.083707711],[0,0,0,0],[9E+09,9E+09,9E+09,9E+09,9E+09,9E+09]];
  CONST robtarget Target_720:=[[-222.704839595,1964.209068673,117.380213056],[0.068473279,-0.432866097,-0.887813704,-0.140446353],[0,0,0,0],[9E+09,9E+09,9E+09,9E+09,9E+09,9E+09]];
  CONST robtarget Target_730:=[[-249.997924122,1997.241230748,129.041491786],[0.079170009,-0.432991998,-0.883269725,-0.161507378],[0,0,0,0],[9E+09,9E+09,9E+09,9E+09,9E+09,9E+09]];
  VAR SyncIdent Ident_1;
  VAR SyncIdent Ident_2;
  PERS Tasks Task_1{2}:=[["T_ROB1"],["T_ROB2"]];
  CONST robtarget pTarget_1:=[[-249.999982853,-2.758889972,70.910184906],[0.218727356,-0.500318169,-0.767608398,-0.335585192],[-1,-1,2,0],[9E+09,9E+09,9E+09,9E+09,9E+09,9E+09]];
  CONST robtarget pTarget_2:=[[-272.861882141,33.004474389,109.271780859],[0.218070089,-0.506815721,-0.766106922,-0.329641389],[0,0,2,0],[9E+09,9E+09,9E+09,9E+09,9E+09,9E+09]];
  CONST robtarget pTarget_3:=[[-293.910897367,69.704818109,146.788417202],[0.216170638,-0.529374655,-0.759500655,-0.31014752],[0,0,2,0],[9E+09,9E+09,9E+09,9E+09,9E+09,9E+09]];
  CONST robtarget pTarget_4:=[[-309.050426556,104.288383302,178.815114444],[0.21342224,-0.572774596,-0.741629436,-0.276343968],[0,0,2,0],[9E+09,9E+09,9E+09,9E+09,9E+09,9E+09]];
  CONST robtarget pTarget_5:=[[-315.825879092,131.080277492,200.511993969],[0.210053721,-0.629622145,-0.709520967,-0.236713724],[0,0,2,0],[9E+09,9E+09,9E+09,9E+09,9E+09,9E+09]];
  CONST robtarget pTarget_6:=[[-316.950658169,142.443127526,208.736277874],[0.207697142,-0.661844648,-0.687247207,-0.215672981],[0,0,2,0],[9E+09,9E+09,9E+09,9E+09,9E+09,9E+09]];
  CONST robtarget pTarget_7:=[[-316.982935585,150.772590841,214.3610347],[0.205252938,-0.688776438,-0.666352974,-0.198574832],[0,0,2,0],[9E+09,9E+09,9E+09,9E+09,9E+09,9E+09]];
  CONST robtarget pTarget_8:=[[-316.205680892,159.554683635,219.903696352],[0.201637265,-0.719895206,-0.63953479,-0.179132795],[0,0,2,0],[9E+09,9E+09,9E+09,9E+09,9E+09,9E+09]];
  CONST robtarget pTarget_9:=[[-312.752948072,174.804783132,228.537464358],[0.190111882,-0.772966578,-0.58777574,-0.144567705],[0,0,2,0],[9E+09,9E+09,9E+09,9E+09,9E+09,9E+09]];
  CONST robtarget pTarget_10:=[[-304.930214203,193.592151989,237.349035256],[0.164735755,-0.829787877,-0.523003524,-0.10383412],[0,0,2,0],[9E+09,9E+09,9E+09,9E+09,9E+09,9E+09]];
  CONST robtarget pTarget_11:=[[-295.354295578,209.583594983,243.175290065],[0.133385277,-0.8681553,-0.472487419,-0.0725974],[0,0,2,0],[9E+09,9E+09,9E+09,9E+09,9E+09,9E+09]];
  CONST robtarget pTarget_12:=[[-283.899433589,224.892894657,247.248273661],[0.09596897,-0.895792145,-0.43151926,-0.046233299],[0,0,2,0],[9E+09,9E+09,9E+09,9E+09,9E+09,9E+09]];
  CONST robtarget pTarget_13:=[[-263.241026813,247.749218638,250.55023108],[0.034733915,-0.921371183,-0.386853892,-0.014586439],[0,0,2,0],[9E+09,9E+09,9E+09,9E+09,9E+09,9E+09]];
  CONST robtarget pTarget_14:=[[-240.981922532,269.119698062,250.907521043],[0.018476819,0.931695715,0.362698235,-0.007189718],[0,0,2,0],[9E+09,9E+09,9E+09,9E+09,9E+09,9E+09]];
  CONST robtarget pTarget_15:=[[-208.413183072,298.032091366,247.788399876],[0.079579938,0.931527315,0.353569956,-0.030202349],[0,0,2,0],[9E+09,9E+09,9E+09,9E+09,9E+09,9E+09]];
  CONST robtarget pTarget_16:=[[-176.052193628,326.809908438,241.224111838],[0.12634207,0.919491885,0.3687884,-0.050670216],[0,0,2,0],[9E+09,9E+09,9E+09,9E+09,9E+09,9E+09]];
  CONST robtarget pTarget_17:=[[-156.253006236,345.812062065,235.319898524],[0.149532826,0.905306343,0.392253601,-0.0647879],[0,0,2,0],[9E+09,9E+09,9E+09,9E+09,9E+09,9E+09]];
  CONST robtarget pTarget_18:=[[-137.912729763,365.729836666,228.01394112],[0.167326436,0.883813043,0.429269038,-0.081267835],[0,0,2,0],[9E+09,9E+09,9E+09,9E+09,9E+09,9E+09]];
  CONST robtarget pTarget_19:=[[-123.076086452,385.29684741,219.899751042],[0.178122742,0.85378951,0.478888901,-0.099905866],[0,0,2,0],[9E+09,9E+09,9E+09,9E+09,9E+09,9E+09]];
  CONST robtarget pTarget_20:=[[-112.485109992,403.753339887,211.517517208],[0.182306761,0.816637689,0.534446355,-0.119307265],[0,0,2,0],[9E+09,9E+09,9E+09,9E+09,9E+09,9E+09]];
  CONST robtarget pTarget_21:=[[-105.670178268,420.540737418,203.413907188],[0.182491022,0.780616625,0.582081066,-0.136074774],[0,0,2,0],[9E+09,9E+09,9E+09,9E+09,9E+09,9E+09]];
  CONST robtarget pTarget_22:=[[-101.15368719,437.795748992,194.701831653],[0.179971611,0.74337611,0.626119394,-0.151580612],[0,0,2,0],[9E+09,9E+09,9E+09,9E+09,9E+09,9E+09]];
  CONST robtarget pTarget_23:=[[-99.004909593,453.550262222,186.488207379],[0.175916518,0.71039217,0.661486962,-0.163802752],[0,0,2,0],[9E+09,9E+09,9E+09,9E+09,9E+09,9E+09]];
  CONST robtarget pTarget_24:=[[-98.517183319,465.110586386,180.346452198],[0.172174243,0.687303096,0.684519732,-0.171473672],[0,0,2,0],[9E+09,9E+09,9E+09,9E+09,9E+09,9E+09]];
  CONST robtarget pTarget_25:=[[-98.914532644,477.216281927,173.843762862],[0.167750144,0.664394684,0.706153116,-0.178290128],[0,0,2,0],[9E+09,9E+09,9E+09,9E+09,9E+09,9E+09]];
  CONST robtarget pTarget_26:=[[-101.159356556,495.695093883,163.844728445],[0.160294978,0.632212446,0.734783022,-0.186297754],[0,0,2,0],[9E+09,9E+09,9E+09,9E+09,9E+09,9E+09]];
  CONST robtarget pTarget_27:=[[-106.105437701,517.567072003,152.023011482],[0.150752486,0.598596041,0.762916676,-0.192131759],[0,0,2,0],[9E+09,9E+09,9E+09,9E+09,9E+09,9E+09]];
  CONST robtarget pTarget_28:=[[-113.660661173,540.614926982,139.756423783],[0.140145495,0.568163603,0.787297941,-0.194194007],[0,0,2,0],[9E+09,9E+09,9E+09,9E+09,9E+09,9E+09]];
  CONST robtarget pTarget_29:=[[-130.507634781,578.661910337,120.438432349],[0.121655696,0.527679401,0.819198584,-0.188859792],[0,0,2,0],[9E+09,9E+09,9E+09,9E+09,9E+09,9E+09]];
  CONST robtarget pTarget_30:=[[-151.26626902,615.99978174,103.274739393],[0.102156402,0.497611338,0.84376747,-0.173215132],[0,0,2,0],[9E+09,9E+09,9E+09,9E+09,9E+09,9E+09]];
  CONST robtarget pTarget_31:=[[-176.025786598,654.711283406,88.195694778],[0.080012228,0.474620075,0.864351323,-0.1457073],[0,-1,2,0],[9E+09,9E+09,9E+09,9E+09,9E+09,9E+09]];
  CONST robtarget pTarget_32:=[[-202.970062049,693.301100095,76.713070128],[0.055270211,0.458961325,0.880375462,-0.106012978],[0,-1,2,0],[9E+09,9E+09,9E+09,9E+09,9E+09,9E+09]];
  CONST robtarget pTarget_33:=[[-231.601523866,732.417884044,69.538476495],[0.026891104,0.450400962,0.890835711,-0.053174969],[0,-1,2,0],[9E+09,9E+09,9E+09,9E+09,9E+09,9E+09]];
  CONST robtarget pTarget_34:=[[-260.469520449,771.255872105,67.252197805],[0.000040228,0.449762351,0.893148263,-0.000073424],[0,-1,2,0],[9E+09,9E+09,9E+09,9E+09,9E+09,9E+09]];
  CONST robtarget pTarget_35:=[[-291.670914504,813.968978886,69.776506912],[0.026409008,-0.457823003,-0.887175769,-0.051184145],[0,-1,2,0],[9E+09,9E+09,9E+09,9E+09,9E+09,9E+09]];
  CONST robtarget pTarget_36:=[[-321.099734743,856.496080673,76.870467066],[0.050519426,-0.474571222,-0.873828081,-0.093029174],[0,-1,2,0],[9E+09,9E+09,9E+09,9E+09,9E+09,9E+09]];
  CONST robtarget pTarget_37:=[[-347.607513558,898.756689263,87.793598215],[0.073136056,-0.499938347,-0.853878066,-0.124920036],[0,-1,2,0],[9E+09,9E+09,9E+09,9E+09,9E+09,9E+09]];
  CONST robtarget pTarget_38:=[[-370.045783343,940.670316452,101.805420301],[0.094966939,-0.534398849,-0.826923789,-0.146956446],[0,0,2,0],[9E+09,9E+09,9E+09,9E+09,9E+09,9E+09]];
  CONST robtarget pTarget_39:=[[-386.422266732,979.738715708,117.17043925],[0.115288749,-0.575885363,-0.793612764,-0.15888151],[0,0,2,0],[9E+09,9E+09,9E+09,9E+09,9E+09,9E+09]];
  CONST robtarget pTarget_40:=[[-397.441208907,1019.683400433,134.627667281],[0.13626385,-0.628500265,-0.748392037,-0.162261943],[0,0,2,0],[9E+09,9E+09,9E+09,9E+09,9E+09,9E+09]];
  CONST robtarget pTarget_41:=[[-400.684804054,1043.11370182,145.484353571],[0.148540441,-0.664075872,-0.715089643,-0.159955541],[0,0,2,0],[9E+09,9E+09,9E+09,9E+09,9E+09,9E+09]];
  CONST robtarget pTarget_42:=[[-401.329047191,1057.287009915,152.213033994],[0.155841519,-0.687048546,-0.692119904,-0.156996034],[0,0,2,0],[9E+09,9E+09,9E+09,9E+09,9E+09,9E+09]];
  CONST robtarget pTarget_43:=[[-400.962324214,1070.626836833,158.630266332],[0.162306824,-0.708452998,-0.669495106,-0.153385619],[0,0,2,0],[9E+09,9E+09,9E+09,9E+09,9E+09,9E+09]];
  CONST robtarget pTarget_44:=[[-398.849183148,1089.50771848,167.811803441],[0.170245025,-0.736429133,-0.637918276,-0.147475544],[0,0,2,0],[9E+09,9E+09,9E+09,9E+09,9E+09,9E+09]];
  CONST robtarget pTarget_45:=[[-394.2955253,1110.833995661,178.254456324],[0.177319257,-0.764612398,-0.603598072,-0.139982605],[0,0,2,0],[9E+09,9E+09,9E+09,9E+09,9E+09,9E+09]];
  CONST robtarget pTarget_46:=[[-380.757471944,1149.009379517,196.873180768],[0.184540979,-0.806336545,-0.547767283,-0.125367489],[0,0,2,0],[9E+09,9E+09,9E+09,9E+09,9E+09,9E+09]];
  CONST robtarget pTarget_47:=[[-357.502459174,1192.924465348,217.59618262],[0.183790476,-0.842562217,-0.494638737,-0.107900377],[0,0,2,0],[9E+09,9E+09,9E+09,9E+09,9E+09,9E+09]];
  CONST robtarget pTarget_48:=[[-328.871131996,1234.787325405,235.977961384],[0.173717681,-0.868301552,-0.455593953,-0.091152247],[0,0,2,0],[9E+09,9E+09,9E+09,9E+09,9E+09,9E+09]];
  CONST robtarget pTarget_49:=[[-297.082271262,1274.589016917,251.512758604],[0.155168267,-0.886933809,-0.428543903,-0.074975664],[0,0,2,0],[9E+09,9E+09,9E+09,9E+09,9E+09,9E+09]];
  CONST robtarget pTarget_50:=[[-262.487284271,1314.072540843,264.392414029],[0.127341788,-0.900832553,-0.410985687,-0.05809945],[0,0,2,0],[9E+09,9E+09,9E+09,9E+09,9E+09,9E+09]];
  CONST robtarget pTarget_51:=[[-226.57533141,1353.20491494,273.985918464],[0.089566851,-0.910054777,-0.40274885,-0.039641474],[0,0,2,0],[9E+09,9E+09,9E+09,9E+09,9E+09,9E+09]];
  CONST robtarget pTarget_52:=[[-190.835573063,1391.953156962,279.66226271],[0.041472362,-0.913491552,-0.404321853,-0.018359371],[0,0,2,0],[9E+09,9E+09,9E+09,9E+09,9E+09,9E+09]];
  CONST robtarget pTarget_53:=[[-154.17838296,1433.251807008,280.664288166],[0.021076524,0.908000293,0.418326405,-0.009709151],[0,0,2,0],[9E+09,9E+09,9E+09,9E+09,9E+09,9E+09]];
  CONST robtarget pTarget_54:=[[-136.486765374,1454.464402311,278.839431135],[0.056847305,0.900059217,0.431184714,-0.027231083],[0,0,2,0],[9E+09,9E+09,9E+09,9E+09,9E+09,9E+09]];
  CONST robtarget pTarget_55:=[[-119.667936085,1475.943296051,275.178359687],[0.094528682,0.887510172,0.448451627,-0.047761511],[0,0,2,0],[9E+09,9E+09,9E+09,9E+09,9E+09,9E+09]];
  CONST robtarget pTarget_56:=[[-95.234012575,1510.930409762,264.895769368],[0.154652239,0.855971808,0.485490887,-0.087712866],[0,0,2,0],[9E+09,9E+09,9E+09,9E+09,9E+09,9E+09]];
  CONST robtarget pTarget_57:=[[-75.878773781,1544.776154817,249.922804533],[0.194530976,0.816269054,0.529114868,-0.126095149],[0,0,2,0],[9E+09,9E+09,9E+09,9E+09,9E+09,9E+09]];
  CONST robtarget pTarget_58:=[[-61.453141161,1578.970333156,230.887297549],[0.213995385,0.770545603,0.578493801,-0.160656062],[0,0,2,0],[9E+09,9E+09,9E+09,9E+09,9E+09,9E+09]];
  CONST robtarget pTarget_59:=[[-52.708491627,1614.593802629,208.278633282],[0.2154784,0.717600683,0.634304305,-0.190463561],[0,0,2,0],[9E+09,9E+09,9E+09,9E+09,9E+09,9E+09]];
  CONST robtarget pTarget_60:=[[-50.933702908,1632.587902032,196.272906508],[0.21049827,0.690275184,0.662147881,-0.201917887],[0,0,2,0],[9E+09,9E+09,9E+09,9E+09,9E+09,9E+09]];
  CONST robtarget pTarget_61:=[[-50.773310022,1647.959263114,185.915184413],[0.204128011,0.668216161,0.684203386,-0.209008715],[0,0,2,0],[9E+09,9E+09,9E+09,9E+09,9E+09,9E+09]];
  CONST robtarget pTarget_62:=[[-52.133848077,1666.482662645,173.501879979],[0.194191907,0.643165566,0.709079002,-0.214089997],[0,0,2,0],[9E+09,9E+09,9E+09,9E+09,9E+09,9E+09]];
  CONST robtarget pTarget_63:=[[-58.782669223,1700.877359567,151.375731817],[0.170010517,0.600573609,0.751746936,-0.2128011],[0,0,2,0],[9E+09,9E+09,9E+09,9E+09,9E+09,9E+09]];
  CONST robtarget pTarget_64:=[[-65.573382217,1722.873059911,138.379981308],[0.151037739,0.575542272,0.777381463,-0.204001853],[0,0,2,0],[9E+09,9E+09,9E+09,9E+09,9E+09,9E+09]];
  CONST robtarget pTarget_65:=[[-74.172458436,1744.953551809,126.646734635],[0.129487963,0.551841007,0.802051755,-0.188194988],[0,0,2,0],[9E+09,9E+09,9E+09,9E+09,9E+09,9E+09]];
  CONST robtarget pTarget_66:=[[-84.216406288,1766.689925652,116.694082829],[0.10605041,0.529831854,0.825081517,-0.165142384],[0,0,2,0],[9E+09,9E+09,9E+09,9E+09,9E+09,9E+09]];
  CONST robtarget pTarget_67:=[[-95.703735197,1788.481494933,108.58929655],[0.080632832,0.509232536,0.84630056,-0.133999749],[-1,0,2,0],[9E+09,9E+09,9E+09,9E+09,9E+09,9E+09]];
  CONST robtarget pTarget_68:=[[-107.611560112,1808.886865418,102.932793062],[0.055430058,0.491624274,0.863570533,-0.097360244],[-1,-1,2,0],[9E+09,9E+09,9E+09,9E+09,9E+09,9E+09]];
  CONST robtarget pTarget_69:=[[-120.619803812,1829.451884245,99.303968751],[0.029389138,0.476040843,0.877262115,-0.054153266],[-1,-1,2,0],[9E+09,9E+09,9E+09,9E+09,9E+09,9E+09]];
  CONST robtarget pTarget_70:=[[-148.697947715,1869.907233475,98.051310221],[0.01238213,-0.453317439,-0.890930671,-0.024341782],[-1,-1,2,0],[9E+09,9E+09,9E+09,9E+09,9E+09,9E+09]];
  CONST robtarget pTarget_71:=[[-178.285867762,1909.003244069,102.928222428],[0.041270541,-0.440304957,-0.892984494,-0.083707711],[-1,-1,2,0],[9E+09,9E+09,9E+09,9E+09,9E+09,9E+09]];
  CONST robtarget pTarget_72:=[[-222.704839595,1964.209068673,117.380213056],[0.068473279,-0.432866097,-0.887813704,-0.140446353],[-1,-1,2,0],[9E+09,9E+09,9E+09,9E+09,9E+09,9E+09]];
  CONST robtarget pTarget_73:=[[-249.997924122,1997.241230748,129.041491786],[0.079170009,-0.432991998,-0.883269725,-0.161507378],[-1,-1,2,0],[9E+09,9E+09,9E+09,9E+09,9E+09,9E+09]];
  CONST jointtarget p1600_Home:=[[-0.000000291,-39.999998836,0.000001581,0.000002251,25.000000127,180.000018669],[9E+09,9E+09,9E+09,9E+09,9E+09,9E+09]];
  PROC Path_process()
    MoveL Target_10,v200,z1,tWeldGun\WObj:=obWorkpiece;
    MoveL Target_20,v200,z1,tWeldGun\WObj:=obWorkpiece;
    MoveL Target_30,v200,z1,tWeldGun\WObj:=obWorkpiece;
    MoveL Target_40,v200,z1,tWeldGun\WObj:=obWorkpiece;
    MoveL Target_50,v200,z1,tWeldGun\WObj:=obWorkpiece;
    MoveL Target_60,v200,z1,tWeldGun\WObj:=obWorkpiece;
    MoveL Target_70,v200,z1,tWeldGun\WObj:=obWorkpiece;
    MoveL Target_80,v200,z1,tWeldGun\WObj:=obWorkpiece;
    MoveL Target_90,v200,z1,tWeldGun\WObj:=obWorkpiece;
    MoveL Target_100,v200,z1,tWeldGun\WObj:=obWorkpiece;
    MoveL Target_110,v200,z1,tWeldGun\WObj:=obWorkpiece;
    MoveL Target_120,v200,z1,tWeldGun\WObj:=obWorkpiece;
    MoveL Target_130,v200,z1,tWeldGun\WObj:=obWorkpiece;
    MoveL Target_140,v200,z1,tWeldGun\WObj:=obWorkpiece;
    MoveL Target_150,v200,z1,tWeldGun\WObj:=obWorkpiece;
    MoveL Target_160,v200,z1,tWeldGun\WObj:=obWorkpiece;
    MoveL Target_170,v200,z1,tWeldGun\WObj:=obWorkpiece;
    MoveL Target_180,v200,z1,tWeldGun\WObj:=obWorkpiece;
    MoveL Target_190,v200,z1,tWeldGun\WObj:=obWorkpiece;
    MoveL Target_200,v200,z1,tWeldGun\WObj:=obWorkpiece;
    MoveL Target_210,v200,z1,tWeldGun\WObj:=obWorkpiece;
    MoveL Target_220,v200,z1,tWeldGun\WObj:=obWorkpiece;
    MoveL Target_230,v200,z1,tWeldGun\WObj:=obWorkpiece;
    MoveL Target_240,v200,z1,tWeldGun\WObj:=obWorkpiece;
    MoveL Target_250,v200,z1,tWeldGun\WObj:=obWorkpiece;
    MoveL Target_260,v200,z1,tWeldGun\WObj:=obWorkpiece;
    MoveL Target_270,v200,z1,tWeldGun\WObj:=obWorkpiece;
    MoveL Target_280,v200,z1,tWeldGun\WObj:=obWorkpiece;
    MoveL Target_290,v200,z1,tWeldGun\WObj:=obWorkpiece;
    MoveL Target_300,v200,z1,tWeldGun\WObj:=obWorkpiece;
    MoveL Target_310,v200,z1,tWeldGun\WObj:=obWorkpiece;
    MoveL Target_320,v200,z1,tWeldGun\WObj:=obWorkpiece;
    MoveL Target_330,v200,z1,tWeldGun\WObj:=obWorkpiece;
    MoveL Target_340,v200,z1,tWeldGun\WObj:=obWorkpiece;
    MoveL Target_350,v200,z1,tWeldGun\WObj:=obWorkpiece;
    MoveL Target_360,v200,z1,tWeldGun\WObj:=obWorkpiece;
    MoveL Target_370,v200,z1,tWeldGun\WObj:=obWorkpiece;
    MoveL Target_380,v200,z1,tWeldGun\WObj:=obWorkpiece;
    MoveL Target_390,v200,z1,tWeldGun\WObj:=obWorkpiece;
    MoveL Target_400,v200,z1,tWeldGun\WObj:=obWorkpiece;
    MoveL Target_410,v200,z1,tWeldGun\WObj:=obWorkpiece;
    MoveL Target_420,v200,z1,tWeldGun\WObj:=obWorkpiece;
    MoveL Target_430,v200,z1,tWeldGun\WObj:=obWorkpiece;
    MoveL Target_440,v200,z1,tWeldGun\WObj:=obWorkpiece;
    MoveL Target_450,v200,z1,tWeldGun\WObj:=obWorkpiece;
    MoveL Target_460,v200,z1,tWeldGun\WObj:=obWorkpiece;
    MoveL Target_470,v200,z1,tWeldGun\WObj:=obWorkpiece;
    MoveL Target_480,v200,z1,tWeldGun\WObj:=obWorkpiece;
    MoveL Target_490,v200,z1,tWeldGun\WObj:=obWorkpiece;
    MoveL Target_500,v200,z1,tWeldGun\WObj:=obWorkpiece;
    MoveL Target_510,v200,z1,tWeldGun\WObj:=obWorkpiece;
    MoveL Target_520,v200,z1,tWeldGun\WObj:=obWorkpiece;
    MoveL Target_530,v200,z1,tWeldGun\WObj:=obWorkpiece;
    MoveL Target_540,v200,z1,tWeldGun\WObj:=obWorkpiece;
    MoveL Target_550,v200,z1,tWeldGun\WObj:=obWorkpiece;
    MoveL Target_560,v200,z1,tWeldGun\WObj:=obWorkpiece;
    MoveL Target_570,v200,z1,tWeldGun\WObj:=obWorkpiece;
    MoveL Target_580,v200,z1,tWeldGun\WObj:=obWorkpiece;
    MoveL Target_590,v200,z1,tWeldGun\WObj:=obWorkpiece;
    MoveL Target_600,v200,z1,tWeldGun\WObj:=obWorkpiece;
    MoveL Target_610,v200,z1,tWeldGun\WObj:=obWorkpiece;
    MoveL Target_620,v200,z1,tWeldGun\WObj:=obWorkpiece;
    MoveL Target_630,v200,z1,tWeldGun\WObj:=obWorkpiece;
    MoveL Target_640,v200,z1,tWeldGun\WObj:=obWorkpiece;
    MoveL Target_650,v200,z1,tWeldGun\WObj:=obWorkpiece;
    MoveL Target_660,v200,z1,tWeldGun\WObj:=obWorkpiece;
    MoveL Target_670,v200,z1,tWeldGun\WObj:=obWorkpiece;
    MoveL Target_680,v200,z1,tWeldGun\WObj:=obWorkpiece;
    MoveL Target_690,v200,z1,tWeldGun\WObj:=obWorkpiece;
    MoveL Target_700,v200,z1,tWeldGun\WObj:=obWorkpiece;
    MoveL Target_710,v200,z1,tWeldGun\WObj:=obWorkpiece;
    MoveL Target_720,v200,z1,tWeldGun\WObj:=obWorkpiece;
    MoveL Target_730,v200,z1,tWeldGun\WObj:=obWorkpiece;
  ENDPROC
  PROC mmPath_1()
    MoveAbsJ p1600_Home,v1000,z100,tool0\WObj:=wobj0;
    SyncMoveOn Ident_1,Task_1;
    MoveJ pTarget_1\ID:=10,v200,z1,tWeldGun\WObj:=obWorkpiece;
    MoveL pTarget_2\ID:=20,v200,z1,tWeldGun\WObj:=obWorkpiece;
    MoveL pTarget_3\ID:=30,v200,z1,tWeldGun\WObj:=obWorkpiece;
    MoveL pTarget_4\ID:=40,v200,z1,tWeldGun\WObj:=obWorkpiece;
    MoveL pTarget_5\ID:=50,v200,z1,tWeldGun\WObj:=obWorkpiece;
    MoveL pTarget_6\ID:=60,v200,z1,tWeldGun\WObj:=obWorkpiece;
    MoveL pTarget_7\ID:=70,v200,z1,tWeldGun\WObj:=obWorkpiece;
    MoveL pTarget_8\ID:=80,v200,z1,tWeldGun\WObj:=obWorkpiece;
    MoveL pTarget_9\ID:=90,v200,z1,tWeldGun\WObj:=obWorkpiece;
    MoveL pTarget_10\ID:=100,v200,z1,tWeldGun\WObj:=obWorkpiece;
    MoveL pTarget_11\ID:=110,v200,z1,tWeldGun\WObj:=obWorkpiece;
    MoveL pTarget_12\ID:=120,v200,z1,tWeldGun\WObj:=obWorkpiece;
    MoveL pTarget_13\ID:=130,v200,z1,tWeldGun\WObj:=obWorkpiece;
    MoveL pTarget_14\ID:=140,v200,z1,tWeldGun\WObj:=obWorkpiece;
    MoveL pTarget_15\ID:=150,v200,z1,tWeldGun\WObj:=obWorkpiece;
    MoveL pTarget_16\ID:=160,v200,z1,tWeldGun\WObj:=obWorkpiece;
    MoveL pTarget_17\ID:=170,v200,z1,tWeldGun\WObj:=obWorkpiece;
    MoveL pTarget_18\ID:=180,v200,z1,tWeldGun\WObj:=obWorkpiece;
    MoveL pTarget_19\ID:=190,v200,z1,tWeldGun\WObj:=obWorkpiece;
    MoveL pTarget_20\ID:=200,v200,z1,tWeldGun\WObj:=obWorkpiece;
    MoveL pTarget_21\ID:=210,v200,z1,tWeldGun\WObj:=obWorkpiece;
    MoveL pTarget_22\ID:=220,v200,z1,tWeldGun\WObj:=obWorkpiece;
    MoveL pTarget_23\ID:=230,v200,z1,tWeldGun\WObj:=obWorkpiece;
    MoveL pTarget_24\ID:=240,v200,z1,tWeldGun\WObj:=obWorkpiece;
    MoveL pTarget_25\ID:=250,v200,z1,tWeldGun\WObj:=obWorkpiece;
    MoveL pTarget_26\ID:=260,v200,z1,tWeldGun\WObj:=obWorkpiece;
    MoveL pTarget_27\ID:=270,v200,z1,tWeldGun\WObj:=obWorkpiece;
    MoveL pTarget_28\ID:=280,v200,z1,tWeldGun\WObj:=obWorkpiece;
    MoveL pTarget_29\ID:=290,v200,z1,tWeldGun\WObj:=obWorkpiece;
    MoveL pTarget_30\ID:=300,v200,z1,tWeldGun\WObj:=obWorkpiece;
    MoveL pTarget_31\ID:=310,v200,z1,tWeldGun\WObj:=obWorkpiece;
    MoveL pTarget_32\ID:=320,v200,z1,tWeldGun\WObj:=obWorkpiece;
    MoveL pTarget_33\ID:=330,v200,z1,tWeldGun\WObj:=obWorkpiece;
    MoveL pTarget_34\ID:=340,v200,z1,tWeldGun\WObj:=obWorkpiece;
    MoveL pTarget_35\ID:=350,v200,z1,tWeldGun\WObj:=obWorkpiece;
    MoveL pTarget_36\ID:=360,v200,z1,tWeldGun\WObj:=obWorkpiece;
    MoveL pTarget_37\ID:=370,v200,z1,tWeldGun\WObj:=obWorkpiece;
    MoveL pTarget_38\ID:=380,v200,z1,tWeldGun\WObj:=obWorkpiece;
    MoveL pTarget_39\ID:=390,v200,z1,tWeldGun\WObj:=obWorkpiece;
    MoveL pTarget_40\ID:=400,v200,z1,tWeldGun\WObj:=obWorkpiece;
    MoveL pTarget_41\ID:=410,v200,z1,tWeldGun\WObj:=obWorkpiece;
    MoveL pTarget_42\ID:=420,v200,z1,tWeldGun\WObj:=obWorkpiece;
    MoveL pTarget_43\ID:=430,v200,z1,tWeldGun\WObj:=obWorkpiece;
    MoveL pTarget_44\ID:=440,v200,z1,tWeldGun\WObj:=obWorkpiece;
    MoveL pTarget_45\ID:=450,v200,z1,tWeldGun\WObj:=obWorkpiece;
    MoveL pTarget_46\ID:=460,v200,z1,tWeldGun\WObj:=obWorkpiece;
    MoveL pTarget_47\ID:=470,v200,z1,tWeldGun\WObj:=obWorkpiece;
    MoveL pTarget_48\ID:=480,v200,z1,tWeldGun\WObj:=obWorkpiece;
    MoveL pTarget_49\ID:=490,v200,z1,tWeldGun\WObj:=obWorkpiece;
    MoveL pTarget_50\ID:=500,v200,z1,tWeldGun\WObj:=obWorkpiece;
    MoveL pTarget_51\ID:=510,v200,z1,tWeldGun\WObj:=obWorkpiece;
    MoveL pTarget_52\ID:=520,v200,z1,tWeldGun\WObj:=obWorkpiece;
    MoveL pTarget_53\ID:=530,v200,z1,tWeldGun\WObj:=obWorkpiece;
    MoveL pTarget_54\ID:=540,v200,z1,tWeldGun\WObj:=obWorkpiece;
    MoveL pTarget_55\ID:=550,v200,z1,tWeldGun\WObj:=obWorkpiece;
    MoveL pTarget_56\ID:=560,v200,z1,tWeldGun\WObj:=obWorkpiece;
    MoveL pTarget_57\ID:=570,v200,z1,tWeldGun\WObj:=obWorkpiece;
    MoveL pTarget_58\ID:=580,v200,z1,tWeldGun\WObj:=obWorkpiece;
    MoveL pTarget_59\ID:=590,v200,z1,tWeldGun\WObj:=obWorkpiece;
    MoveL pTarget_60\ID:=600,v200,z1,tWeldGun\WObj:=obWorkpiece;
    MoveL pTarget_61\ID:=610,v200,z1,tWeldGun\WObj:=obWorkpiece;
    MoveL pTarget_62\ID:=620,v200,z1,tWeldGun\WObj:=obWorkpiece;
    MoveL pTarget_63\ID:=630,v200,z1,tWeldGun\WObj:=obWorkpiece;
    MoveL pTarget_64\ID:=640,v200,z1,tWeldGun\WObj:=obWorkpiece;
    MoveL pTarget_65\ID:=650,v200,z1,tWeldGun\WObj:=obWorkpiece;
    MoveL pTarget_66\ID:=660,v200,z1,tWeldGun\WObj:=obWorkpiece;
    MoveL pTarget_67\ID:=670,v200,z1,tWeldGun\WObj:=obWorkpiece;
    MoveL pTarget_68\ID:=680,v200,z1,tWeldGun\WObj:=obWorkpiece;
    MoveL pTarget_69\ID:=690,v200,z1,tWeldGun\WObj:=obWorkpiece;
    MoveL pTarget_70\ID:=700,v200,z1,tWeldGun\WObj:=obWorkpiece;
    MoveL pTarget_71\ID:=710,v200,z1,tWeldGun\WObj:=obWorkpiece;
    MoveL pTarget_72\ID:=720,v200,z1,tWeldGun\WObj:=obWorkpiece;
    MoveL pTarget_73\ID:=730,v200,fine,tWeldGun\WObj:=obWorkpiece;
    SyncMoveOff Ident_2;
    MoveAbsJ p1600_Home,v1000,z100,tool0\WObj:=wobj0;
  ENDPROC
  PROC main()
    mmPath_1;
  ENDPROC
ENDMODULE

